FUNCTION_BLOCK BaseCarrier EXTENDS BaseComponent
VAR_INPUT
END_VAR
VAR_OUTPUT
END_VAR
VAR
	Motor : Motor;
END_VAR

END_FUNCTION_BLOCK

(* stored: Version 1.1.0.1, ProductVersion 3.1.4024.9
   POU BaseCarrier: Id {b216d8a6-3a8b-483a-806a-2347eb7ec6e4}, SpecialFunc None *)
